PROGRAM JIG005_BMW_MGU
VAR
END_VAR

END_PROGRAM

(* stored: Version 1.1.0.1, ProductVersion 3.1.4022.18
   POU JIG005_BMW_MGU: Id {f2c4ef82-5da5-4c7c-bcdd-a2559f874752}, SpecialFunc None *)
